{attribute 'linkalways'} 
{attribute 'no_explicit_call' := 'This FB is a CLASS and must be accessed using methods or properties'}
{attribute 'enable_dynamic_creation'}
FUNCTION_BLOCK FINAL ADD_BYTE EXTENDS Node
VAR
	in1 : _BYTE(0);
	in2 : _BYTE(0);
	out : _BYTE(0);
END_VAR

METHOD PUBLIC Clone : I_Node
VAR
	pNode : POINTER TO ADD_BYTE;
END_VAR
pNode := __NEW(ADD_BYTE);
Clone := pNode^;
END_METHOD

METHOD FB_init : BOOL
VAR_INPUT
	bInitRetains : BOOL; // if TRUE, the retain variables are initialized (warm start / cold start)
	bInCopyCode : BOOL;  // if TRUE, the instance afterwards gets moved into the copy code (online change)
END_VAR
AddInput('in1',THIS^.in1);
AddInput('in2',THIS^.in2);
AddOutput('out', THIS^.out);
END_METHOD

METHOD PROTECTED OnExecute
VAR
END_VAR
out.Value := in1.Value + in2.Value;
END_METHOD

END_FUNCTION_BLOCK

(* stored: Version 1.1.0.1, ProductVersion 3.1.4024.15
   POU ADD_BYTE: Id {d1029b3e-80c6-41fb-a3af-870e6b7e132a}, SpecialFunc None
   Folder Constructor: Id {e1a335bf-0736-4d75-a77f-9d345198ef5e}
   Method Clone: Id {4ced6d08-b3f0-4a26-9904-8cce82312d97}
   Method FB_init: Id {9c27a1b2-4b7f-4998-a6d0-f61cd5778963}
   Method OnExecute: Id {097dfb85-871b-4fd9-b8be-da9390c90d6e} *)
